// TIA Portal V16 export
// export: Created 2024-12-03T15:41:45.4867103Z, ExportSetting WithReadOnly, DisplayName Totally Integrated Automation Portal, DisplayVersion V16 Update 6, DisplayName TIA Portal Version Control Interface, DisplayVersion V16 Update 2, DisplayName TIA Portal Openness, DisplayVersion V16 Update 6, DisplayName TIA Portal Teamcenter Gateway, DisplayVersion V16, DisplayName SINAMICS Startdrive Advanced, DisplayVersion V16 Update 5, DisplayName SINAMICS Startdrive G130, G150, S120, S150, SINAMICS MV, S210, DisplayVersion V16 Update 5, DisplayName SINAMICS Startdrive G110M, G120, G120C, G120D, G120P, G115D, DisplayVersion V16 Update 5, DisplayName STEP 7 Professional, DisplayVersion V16 Update 6, DisplayName STEP 7 Safety, DisplayVersion V16, DisplayName WinCC Advanced / Unified PC, DisplayVersion V16 Update 6
TYPE "G120D_SINAPOS_UDT"
// stored: CreationDate 2022-02-10T10:30:20.6863124Z, InterfaceModifiedDate 2021-11-16T12:48:53.5053392Z, IsConsistent true, LibraryConformanceStatus The object is library-conformant., ModifiedDate 2021-11-16T12:48:53.5053392Z
   STRUCT
      Cmd : Struct   // MotorCommands
         Reset : Bool;
         auto : Struct
            mode : Int;
            speed : Real;
            pos : Real;
            enable : Bool;
            direction : Bool;
            executeMode : Bool;
         END_STRUCT;
         manual : Struct
            speed : Real;
            stop : "HandShake_UDT";
            jog1 : "HeartBeatButton_UDT";
            jog2 : "HeartBeatButton_UDT";
            activateHoming { S7_SetPoint := 'True'} : Bool;
         END_STRUCT;
      END_STRUCT;
      Faults : Struct
         status : Word;
         FaultCode : Word;
         FaultActive : Bool;
         Disconnected : Bool;   // The device is not connected
         NotOnTImedOut : Bool;   // Motor not on in time
         NotReady : Bool;
         SafetyProx_1 : Bool;
         SafetyProx_2 : Bool;
         STO_ACTIVE : Bool;
         SAFETY_FAULT_ACTIVE : Bool;
      END_STRUCT;
      Alarms : Struct
         Status : Word;
         AlarmCode : Word;
         AlarmFromDrive : Bool;   // Error from drive
         NotHomed : Bool;
      END_STRUCT;
      Status : Struct
         CurrentMode : Int;
         CmdRunManualActive : Bool;
         Interlocked : Bool;
         ManualModeActive : Bool;
         ManualCommandsDisabled : Bool;
         Running : Bool;
         ActualSpeed : Real;
         ActualPosition : Real;
         ActualDirection : Bool;   // 0 right | 1 left
         atPosition : Bool;
         homed : Bool;
         enabled : Bool;
      END_STRUCT;
      Settings : Struct
         VelocityOverride : Int;   // Velocity override for all operating modes effective: 0-199%
         AccelerationOverride : Int;   // Acceleration override effective 0-100%
         DeaccelarationOverride : Int;   // Deceleration override effective 0-100%
         maxJogSpeed : Int := 10;
         minJogSpeed : Int := 5;
      END_STRUCT;
      Zone : Int;
      info : "MotorInfo";
   END_STRUCT;
END_TYPE
